FUNCTION_BLOCK Production_Runtime_Values
VAR_INPUT
	RT_Started:BOOL;
	Downtime_Signal:BOOL;
	CurrentCPM:REAL;
	ProdStandard:REAL;
	Can_Counter:BOOL;
	
END_VAR
VAR_OUTPUT

	Optimization_Value:REAL;
	CanCount:REAL;
	Uptime_Total_Seconds: DINT;
	Downtime_Total_Seconds: DINT;
	CPM_AVG: REAL;
END_VAR
VAR
	CanCounter: CTU;
	CanCounterMultiplier: CTU;
	CanMultiplierCount: WORD;

	CanCountCurrent: WORD;
	CurrentCanCount: INT;
	Multiplier_CanCountV: REAL;
	CanCountValueB: INT;
	sc_TotalCanCount: INT;
	RT1: tof;
	RT2: TOF;
	Runtime_Value: CTU;
	Spent_Production_Time: WORD;
	SpentProductionTime: INT;

	AdjustedCPM: INT;
	CansEstimatedToBeRun: REAL;
	Opt_ValueA: REAL;
	Opt_before_10: REAL;
	OPTA: INT;
	CheckDivA: CheckDiv_1;
	Estimated_Cans: REAL;
	OptValue_A: REAL;
	Reset: BOOL;
	VerifyDivider: CheckDiv_1;
	SPTReal: REAL;
	
	Downtime_TimeAccumulator: GetTime_Seconds;
	Uptime_TimeAccumulator: GetTime_Seconds;
END_VAR

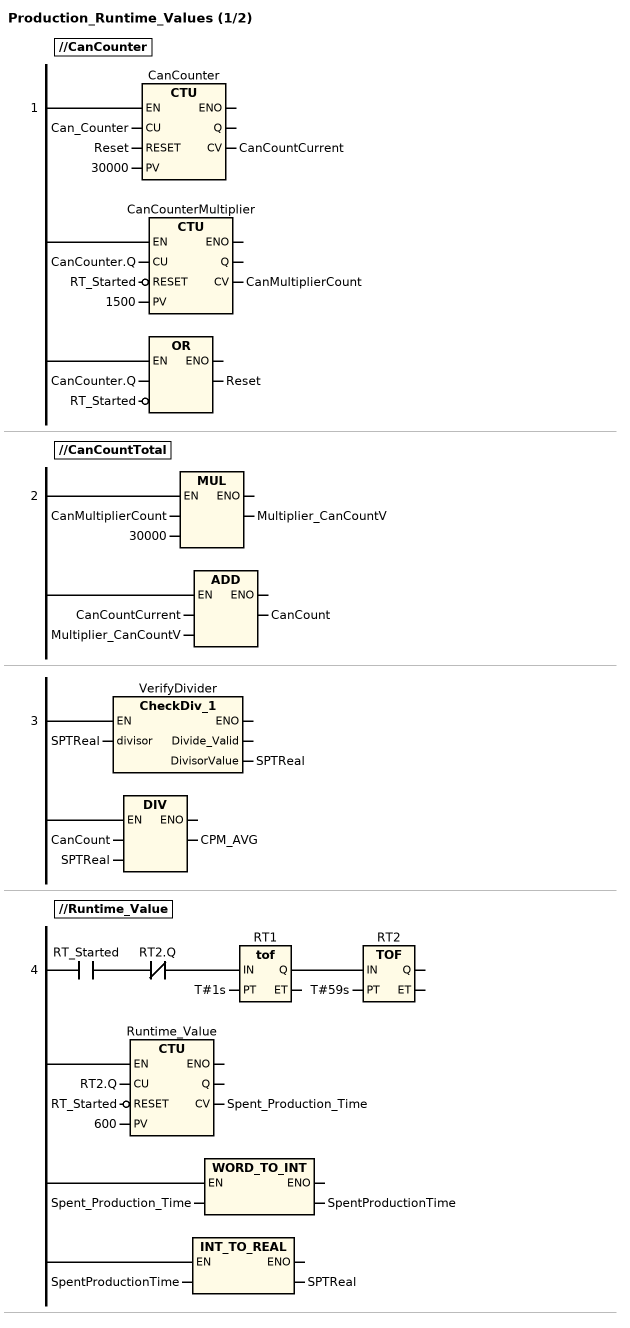
// NETWORK 1
// label: //CanCounter
CanCounter(CU := Can_Counter, RESET := Reset, PV := 30000, CV => CanCountCurrent); // CTU
CanCounterMultiplier(CU := CanCounter.Q, RESET := NOT RT_Started, PV := 1500, CV => CanMultiplierCount); // CTU
Reset := CanCounter.Q OR NOT RT_Started;

// NETWORK 2
// label: //CanCountTotal
Multiplier_CanCountV := CanMultiplierCount * 30000;
CanCount := CanCountCurrent + Multiplier_CanCountV;

// NETWORK 3
VerifyDivider(divisor := SPTReal, DivisorValue => SPTReal); // CheckDiv_1
CPM_AVG := CanCount / SPTReal;

// NETWORK 4
// label: //Runtime_Value
RT1(IN := RT_Started AND NOT RT2.Q, PT := T#1s); // tof
RT2(IN := RT1.Q, PT := T#59s); // TOF
Runtime_Value(CU := RT2.Q, RESET := NOT RT_Started, PV := 600, CV => Spent_Production_Time); // CTU
SpentProductionTime := WORD_TO_INT(Spent_Production_Time);
SPTReal := INT_TO_REAL(SpentProductionTime);

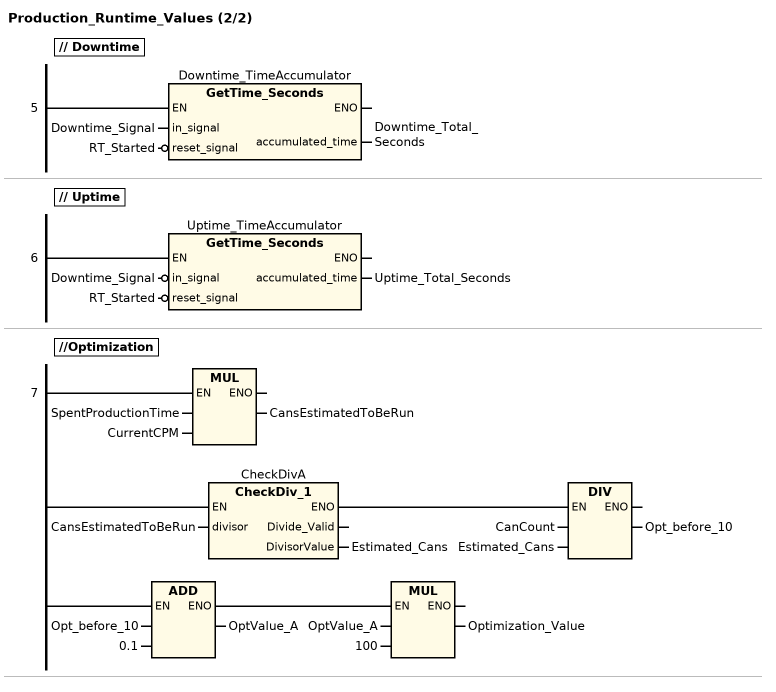
// NETWORK 5
// label: // Downtime
Downtime_TimeAccumulator(
    EN := TRUE,
    in_signal := Downtime_Signal,
    reset_signal := NOT RT_Started,
    accumulated_time => Downtime_Total_Seconds); // GetTime_Seconds

// NETWORK 6
// label: // Uptime
Uptime_TimeAccumulator(
    EN := TRUE,
    in_signal := NOT Downtime_Signal,
    reset_signal := NOT RT_Started,
    accumulated_time => Uptime_Total_Seconds); // GetTime_Seconds

// NETWORK 7
// label: //Optimization
CansEstimatedToBeRun := SpentProductionTime * CurrentCPM;
CheckDivA(divisor := CansEstimatedToBeRun, DivisorValue => Estimated_Cans); // CheckDiv_1
Opt_before_10 := CanCount / Estimated_Cans;
OptValue_A := Opt_before_10 + 0.1;
Optimization_Value := OptValue_A * 100;

END_FUNCTION_BLOCK

(* stored: Version 1.1.0.1, ProductVersion 3.1.4024.15
   POU Production_Runtime_Values: Id {c7ed7983-df8d-463e-81eb-f3a3759191e4}, SpecialFunc None *)
